// TIA Portal V16 export
// export: Created 2021-12-01T20:36:38.1325442Z, ExportSetting WithDefaults, DisplayName Totally Integrated Automation Portal, DisplayVersion V16 Update 4, DisplayName TIA Portal Version Control Interface, DisplayVersion V16 Update 2, DisplayName TIA Portal Openness, DisplayVersion V16 Update 4, DisplayName SINAMICS Startdrive Advanced, DisplayVersion V16 Update 5, DisplayName SINAMICS Startdrive G130, G150, S120, S150, SINAMICS MV, S210, DisplayVersion V16 Update 5, DisplayName SINAMICS Startdrive G110M, G120, G120C, G120D, G120P, G115D, DisplayVersion V16 Update 5, DisplayName STEP 7 Professional, DisplayVersion V16 Update 4, DisplayName STEP 7 Safety, DisplayVersion V16, DisplayName WinCC Advanced, DisplayVersion V16 Update 4
FUNCTION "ST00215_1_FC" : Void   // FC129, LAD
TITLE = ST00215_1
{ S7_Optimized_Access := 'TRUE' }
VERSION : 0.1
// stored: AutoNumber true, IsIECCheckEnabled false, SetENOAutomatically false, UDAEnableTagReadback false
   VAR_IN_OUT
      OPMODE : "OPMODE_OUT_UDT";
      HMI_EXTENSION : "HMI_EXTENSION_PANEL_UDT";
   END_VAR
   VAR_TEMP
      EmptyHS : "RT_HANDSHAKE_UDT";
   END_VAR
BEGIN

REGION Network 1: Alarm
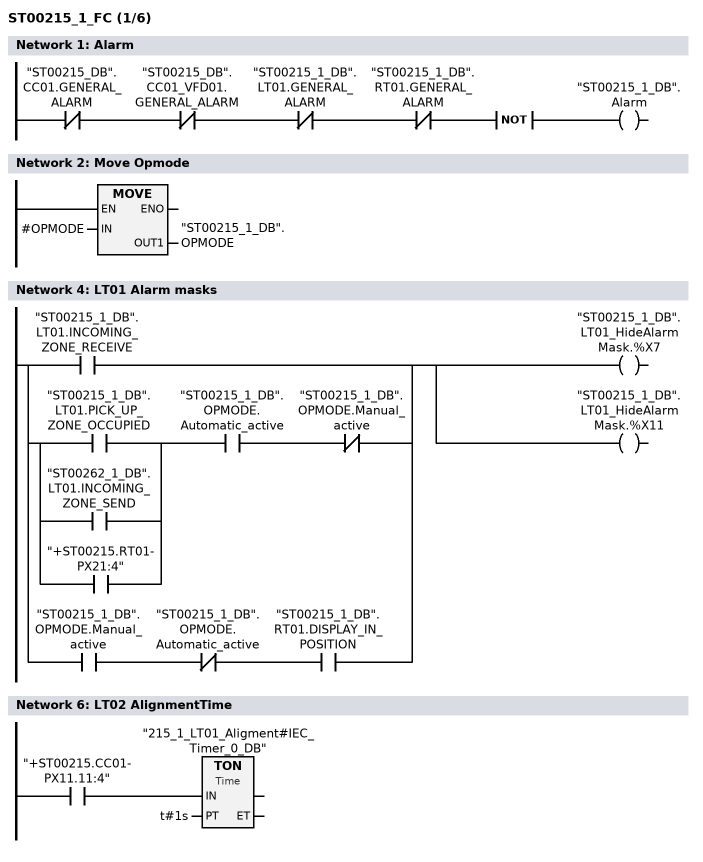
   RUNG wire#powerrail
      I_Contact( "ST00215_DB".CC01.GENERAL_ALARM )
      I_Contact( "ST00215_DB".CC01_VFD01.GENERAL_ALARM )
      I_Contact( "ST00215_1_DB".LT01.GENERAL_ALARM )
      I_Contact( "ST00215_1_DB".RT01.GENERAL_ALARM )
      Not()
      Coil( "ST00215_1_DB".Alarm )
   END_RUNG
   // the same network as SCL:
   "ST00215_1_DB".Alarm := NOT (NOT "ST00215_DB".CC01.GENERAL_ALARM AND NOT "ST00215_DB".CC01_VFD01.GENERAL_ALARM AND NOT "ST00215_1_DB".LT01.GENERAL_ALARM AND NOT "ST00215_1_DB".RT01.GENERAL_ALARM);
END_REGION

REGION Network 2: Move Opmode
   RUNG wire#powerrail
      Move(in := #OPMODE, out1 => "ST00215_1_DB".OPMODE)
   END_RUNG
   // the same network as SCL:
   "ST00215_1_DB".OPMODE := #OPMODE;
END_REGION

REGION Network 3: *******************LT01 Control*******************
END_REGION

REGION Network 4: LT01 Alarm masks
   RUNG wire#powerrail
      Contact( "ST00215_1_DB".LT01.INCOMING_ZONE_RECEIVE )
      wire#w1
      Coil( "ST00215_1_DB".LT01_HideAlarmMask.%X7 )
   END_RUNG
   RUNG wire#powerrail
      Contact( "ST00215_1_DB".LT01.PICK_UP_ZONE_OCCUPIED )
      wire#w2
      Contact( "ST00215_1_DB".OPMODE.Automatic_active )
      I_Contact( "ST00215_1_DB".OPMODE.Manual_active )
   END_RUNG wire#w1
   RUNG wire#powerrail
      Contact( "ST00262_1_DB".LT01.INCOMING_ZONE_SEND )
   END_RUNG wire#w2
   RUNG wire#powerrail
      Contact( "+ST00215.RT01-PX21:4" )
   END_RUNG wire#w2
   RUNG wire#powerrail
      Contact( "ST00215_1_DB".OPMODE.Manual_active )
      I_Contact( "ST00215_1_DB".OPMODE.Automatic_active )
      Contact( "ST00215_1_DB".RT01.DISPLAY_IN_POSITION )
   END_RUNG wire#w1
   RUNG wire#w1
      Coil( "ST00215_1_DB".LT01_HideAlarmMask.%X11 )
   END_RUNG
   // the same network as SCL:
   "ST00215_1_DB".LT01_HideAlarmMask.%X7 := "ST00215_1_DB".LT01.INCOMING_ZONE_RECEIVE OR (("ST00215_1_DB".LT01.PICK_UP_ZONE_OCCUPIED OR "ST00262_1_DB".LT01.INCOMING_ZONE_SEND OR "+ST00215.RT01-PX21:4") AND "ST00215_1_DB".OPMODE.Automatic_active AND NOT "ST00215_1_DB".OPMODE.Manual_active) OR ("ST00215_1_DB".OPMODE.Manual_active AND NOT "ST00215_1_DB".OPMODE.Automatic_active AND "ST00215_1_DB".RT01.DISPLAY_IN_POSITION);
   "ST00215_1_DB".LT01_HideAlarmMask.%X11 := "ST00215_1_DB".LT01_HideAlarmMask.%X7;
END_REGION

REGION Network 5 (SCL): LT01 Parameters
   "ST00215_1_DB".LT01.PARA_SET.Para.HasMidPosition := FALSE;
   "ST00215_1_DB".LT01.PARA_SET.Para.HasRT := true;
   "ST00215_1_DB".LT01.PARA_SET.Para.PosCCStopForward := true;
   "ST00215_1_DB".LT01.PARA_SET.Para.PosCCStopReverse := false;
   "ST00215_1_DB".LT01.PARA_SET.Para.PosRaiseForward_1 := true;
   "ST00215_1_DB".LT01.PARA_SET.Para.PosRaiseForward_2 := true;
   "ST00215_1_DB".LT01.PARA_SET.Para.PosRaiseReverse_1 := true;
   "ST00215_1_DB".LT01.PARA_SET.Para.PosRaiseReverse_2 := false;
   "ST00215_1_DB".LT01.PARA_SET.Para.PosSlowForward := true;
   "ST00215_1_DB".LT01.PARA_SET.Para.PosSlowReverse := false;
   "ST00215_1_DB".LT01.PARA_SET.Set.RuntimeLower := t#10s;
   "ST00215_1_DB".LT01.PARA_SET.Set.RuntimeLift := t#11s;
   "ST00215_1_DB".LT01.PARA_SET.Set.AlignmentTime := t#0ms;
END_REGION

REGION Network 6: LT02 AlignmentTime
   RUNG wire#powerrail
      Contact( "+ST00215.CC01-PX11.11:4" )
      { S7_Templates := "time_type := Time" } "215_1_LT01_Aligment#IEC_Timer_0_DB".TON(pt := t#1s, et =>)
   END_RUNG
   // the same network as SCL:
   "215_1_LT01_Aligment#IEC_Timer_0_DB".TON(IN := "+ST00215.CC01-PX11.11:4", PT := t#1s);
END_REGION

REGION Network 7: LT01 CC Place FB
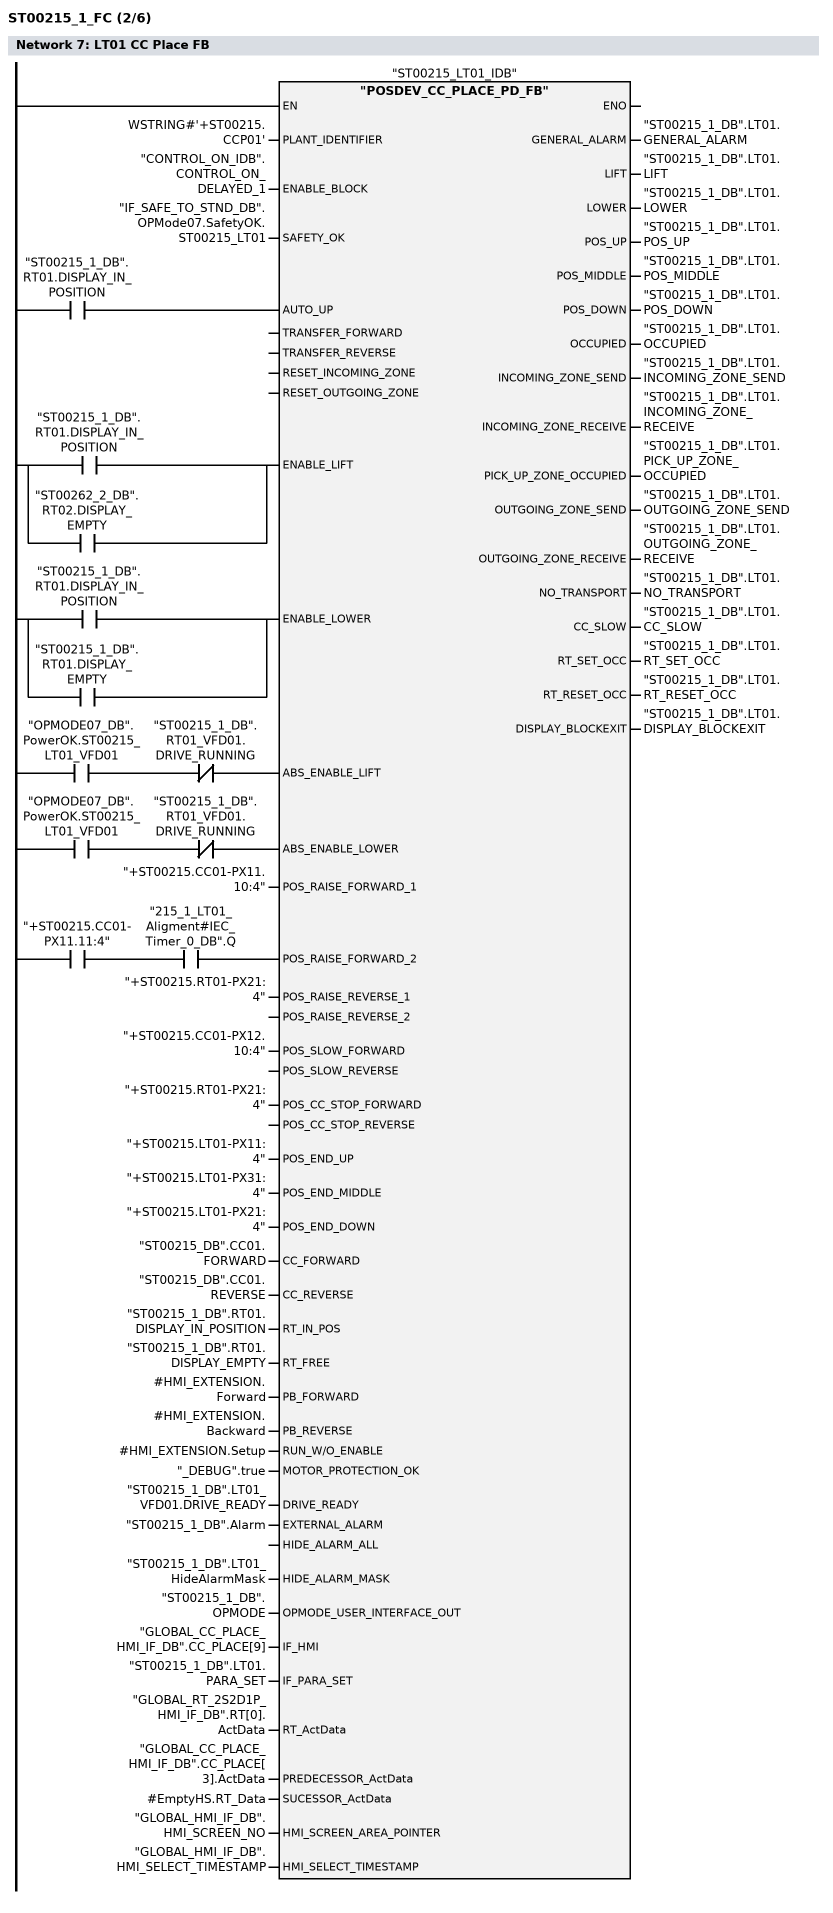
   RUNG wire#powerrail
      "ST00215_LT01_IDB"(AUTO_UP := wire#w1, ENABLE_LIFT := wire#w2, ENABLE_LOWER := wire#w3, ABS_ENABLE_LIFT := wire#w4, ABS_ENABLE_LOWER := wire#w5, POS_RAISE_FORWARD_2 := wire#w6, PLANT_IDENTIFIER := WSTRING#'+ST00215.CCP01', ENABLE_BLOCK := "CONTROL_ON_IDB".CONTROL_ON_DELAYED_1, SAFETY_OK := "IF_SAFE_TO_STND_DB".OPMode07.SafetyOK.ST00215_LT01, TRANSFER_FORWARD :=, TRANSFER_REVERSE :=, RESET_INCOMING_ZONE :=, RESET_OUTGOING_ZONE :=, POS_RAISE_FORWARD_1 := "+ST00215.CC01-PX11.10:4", POS_RAISE_REVERSE_1 := "+ST00215.RT01-PX21:4", POS_RAISE_REVERSE_2 :=, POS_SLOW_FORWARD := "+ST00215.CC01-PX12.10:4", POS_SLOW_REVERSE :=, POS_CC_STOP_FORWARD := "+ST00215.RT01-PX21:4", POS_CC_STOP_REVERSE :=, POS_END_UP := "+ST00215.LT01-PX11:4", POS_END_MIDDLE := "+ST00215.LT01-PX31:4", POS_END_DOWN := "+ST00215.LT01-PX21:4", CC_FORWARD := "ST00215_DB".CC01.FORWARD, CC_REVERSE := "ST00215_DB".CC01.REVERSE, RT_IN_POS := "ST00215_1_DB".RT01.DISPLAY_IN_POSITION, RT_FREE := "ST00215_1_DB".RT01.DISPLAY_EMPTY, PB_FORWARD := #HMI_EXTENSION.Forward, PB_REVERSE := #HMI_EXTENSION.Backward, "RUN_W/O_ENABLE" := #HMI_EXTENSION.Setup, MOTOR_PROTECTION_OK := "_DEBUG".true, DRIVE_READY := "ST00215_1_DB".LT01_VFD01.DRIVE_READY, EXTERNAL_ALARM := "ST00215_1_DB".Alarm, HIDE_ALARM_ALL :=, HIDE_ALARM_MASK := "ST00215_1_DB".LT01_HideAlarmMask, OPMODE_USER_INTERFACE_OUT := "ST00215_1_DB".OPMODE, IF_HMI := "GLOBAL_CC_PLACE_HMI_IF_DB".CC_PLACE[9], IF_PARA_SET := "ST00215_1_DB".LT01.PARA_SET, RT_ActData := "GLOBAL_RT_2S2D1P_HMI_IF_DB".RT[0].ActData, PREDECESSOR_ActData := "GLOBAL_CC_PLACE_HMI_IF_DB".CC_PLACE[3].ActData, SUCESSOR_ActData := #EmptyHS.RT_Data, HMI_SCREEN_AREA_POINTER := "GLOBAL_HMI_IF_DB".HMI_SCREEN_NO, HMI_SELECT_TIMESTAMP := "GLOBAL_HMI_IF_DB".HMI_SELECT_TIMESTAMP, GENERAL_ALARM => "ST00215_1_DB".LT01.GENERAL_ALARM, LIFT => "ST00215_1_DB".LT01.LIFT, LOWER => "ST00215_1_DB".LT01.LOWER, POS_UP => "ST00215_1_DB".LT01.POS_UP, POS_MIDDLE => "ST00215_1_DB".LT01.POS_MIDDLE, POS_DOWN => "ST00215_1_DB".LT01.POS_DOWN, OCCUPIED => "ST00215_1_DB".LT01.OCCUPIED, INCOMING_ZONE_SEND => "ST00215_1_DB".LT01.INCOMING_ZONE_SEND, INCOMING_ZONE_RECEIVE => "ST00215_1_DB".LT01.INCOMING_ZONE_RECEIVE, PICK_UP_ZONE_OCCUPIED => "ST00215_1_DB".LT01.PICK_UP_ZONE_OCCUPIED, OUTGOING_ZONE_SEND => "ST00215_1_DB".LT01.OUTGOING_ZONE_SEND, OUTGOING_ZONE_RECEIVE => "ST00215_1_DB".LT01.OUTGOING_ZONE_RECEIVE, NO_TRANSPORT => "ST00215_1_DB".LT01.NO_TRANSPORT, CC_SLOW => "ST00215_1_DB".LT01.CC_SLOW, RT_SET_OCC => "ST00215_1_DB".LT01.RT_SET_OCC, RT_RESET_OCC => "ST00215_1_DB".LT01.RT_RESET_OCC, DISPLAY_BLOCKEXIT => "ST00215_1_DB".LT01.DISPLAY_BLOCKEXIT)
   END_RUNG
   RUNG wire#powerrail
      Contact( "ST00215_1_DB".RT01.DISPLAY_IN_POSITION )
   END_RUNG wire#w1
   RUNG wire#powerrail
      Contact( "ST00215_1_DB".RT01.DISPLAY_IN_POSITION )
   END_RUNG wire#w2
   RUNG wire#powerrail
      Contact( "ST00262_2_DB".RT02.DISPLAY_EMPTY )
   END_RUNG wire#w2
   RUNG wire#powerrail
      Contact( "ST00215_1_DB".RT01.DISPLAY_IN_POSITION )
   END_RUNG wire#w3
   RUNG wire#powerrail
      Contact( "ST00215_1_DB".RT01.DISPLAY_EMPTY )
   END_RUNG wire#w3
   RUNG wire#powerrail
      Contact( "OPMODE07_DB".PowerOK.ST00215_LT01_VFD01 )
      I_Contact( "ST00215_1_DB".RT01_VFD01.DRIVE_RUNNING )
   END_RUNG wire#w4
   RUNG wire#powerrail
      Contact( "OPMODE07_DB".PowerOK.ST00215_LT01_VFD01 )
      I_Contact( "ST00215_1_DB".RT01_VFD01.DRIVE_RUNNING )
   END_RUNG wire#w5
   RUNG wire#powerrail
      Contact( "+ST00215.CC01-PX11.11:4" )
      Contact( "215_1_LT01_Aligment#IEC_Timer_0_DB".Q )
   END_RUNG wire#w6
   // the same network as SCL:
   "ST00215_LT01_IDB"(PLANT_IDENTIFIER := WSTRING#'+ST00215.CCP01',   // "POSDEV_CC_PLACE_PD_FB"
                      ENABLE_BLOCK := "CONTROL_ON_IDB".CONTROL_ON_DELAYED_1,
                      SAFETY_OK := "IF_SAFE_TO_STND_DB".OPMode07.SafetyOK.ST00215_LT01,
                      AUTO_UP := "ST00215_1_DB".RT01.DISPLAY_IN_POSITION,
                      ENABLE_LIFT := "ST00215_1_DB".RT01.DISPLAY_IN_POSITION OR "ST00262_2_DB".RT02.DISPLAY_EMPTY,
                      ENABLE_LOWER := "ST00215_1_DB".RT01.DISPLAY_IN_POSITION OR "ST00215_1_DB".RT01.DISPLAY_EMPTY,
                      ABS_ENABLE_LIFT := "OPMODE07_DB".PowerOK.ST00215_LT01_VFD01 AND NOT "ST00215_1_DB".RT01_VFD01.DRIVE_RUNNING,
                      ABS_ENABLE_LOWER := "OPMODE07_DB".PowerOK.ST00215_LT01_VFD01 AND NOT "ST00215_1_DB".RT01_VFD01.DRIVE_RUNNING,
                      POS_RAISE_FORWARD_1 := "+ST00215.CC01-PX11.10:4",
                      POS_RAISE_FORWARD_2 := "+ST00215.CC01-PX11.11:4" AND "215_1_LT01_Aligment#IEC_Timer_0_DB".Q,
                      POS_RAISE_REVERSE_1 := "+ST00215.RT01-PX21:4",
                      POS_SLOW_FORWARD := "+ST00215.CC01-PX12.10:4",
                      POS_CC_STOP_FORWARD := "+ST00215.RT01-PX21:4",
                      POS_END_UP := "+ST00215.LT01-PX11:4",
                      POS_END_MIDDLE := "+ST00215.LT01-PX31:4",
                      POS_END_DOWN := "+ST00215.LT01-PX21:4",
                      CC_FORWARD := "ST00215_DB".CC01.FORWARD,
                      CC_REVERSE := "ST00215_DB".CC01.REVERSE,
                      RT_IN_POS := "ST00215_1_DB".RT01.DISPLAY_IN_POSITION,
                      RT_FREE := "ST00215_1_DB".RT01.DISPLAY_EMPTY,
                      PB_FORWARD := #HMI_EXTENSION.Forward,
                      PB_REVERSE := #HMI_EXTENSION.Backward,
                      "RUN_W/O_ENABLE" := #HMI_EXTENSION.Setup,
                      MOTOR_PROTECTION_OK := "_DEBUG".true,
                      DRIVE_READY := "ST00215_1_DB".LT01_VFD01.DRIVE_READY,
                      EXTERNAL_ALARM := "ST00215_1_DB".Alarm,
                      HIDE_ALARM_MASK := "ST00215_1_DB".LT01_HideAlarmMask,
                      OPMODE_USER_INTERFACE_OUT := "ST00215_1_DB".OPMODE,
                      IF_HMI := "GLOBAL_CC_PLACE_HMI_IF_DB".CC_PLACE[9],
                      IF_PARA_SET := "ST00215_1_DB".LT01.PARA_SET,
                      RT_ActData := "GLOBAL_RT_2S2D1P_HMI_IF_DB".RT[0].ActData,
                      PREDECESSOR_ActData := "GLOBAL_CC_PLACE_HMI_IF_DB".CC_PLACE[3].ActData,
                      SUCESSOR_ActData := #EmptyHS.RT_Data,
                      HMI_SCREEN_AREA_POINTER := "GLOBAL_HMI_IF_DB".HMI_SCREEN_NO,
                      HMI_SELECT_TIMESTAMP := "GLOBAL_HMI_IF_DB".HMI_SELECT_TIMESTAMP,
                      GENERAL_ALARM => "ST00215_1_DB".LT01.GENERAL_ALARM,
                      LIFT => "ST00215_1_DB".LT01.LIFT,
                      LOWER => "ST00215_1_DB".LT01.LOWER,
                      POS_UP => "ST00215_1_DB".LT01.POS_UP,
                      POS_MIDDLE => "ST00215_1_DB".LT01.POS_MIDDLE,
                      POS_DOWN => "ST00215_1_DB".LT01.POS_DOWN,
                      OCCUPIED => "ST00215_1_DB".LT01.OCCUPIED,
                      INCOMING_ZONE_SEND => "ST00215_1_DB".LT01.INCOMING_ZONE_SEND,
                      INCOMING_ZONE_RECEIVE => "ST00215_1_DB".LT01.INCOMING_ZONE_RECEIVE,
                      PICK_UP_ZONE_OCCUPIED => "ST00215_1_DB".LT01.PICK_UP_ZONE_OCCUPIED,
                      OUTGOING_ZONE_SEND => "ST00215_1_DB".LT01.OUTGOING_ZONE_SEND,
                      OUTGOING_ZONE_RECEIVE => "ST00215_1_DB".LT01.OUTGOING_ZONE_RECEIVE,
                      NO_TRANSPORT => "ST00215_1_DB".LT01.NO_TRANSPORT,
                      CC_SLOW => "ST00215_1_DB".LT01.CC_SLOW,
                      RT_SET_OCC => "ST00215_1_DB".LT01.RT_SET_OCC,
                      RT_RESET_OCC => "ST00215_1_DB".LT01.RT_RESET_OCC,
                      DISPLAY_BLOCKEXIT => "ST00215_1_DB".LT01.DISPLAY_BLOCKEXIT);
END_REGION

REGION Network 8: LT01 Speed
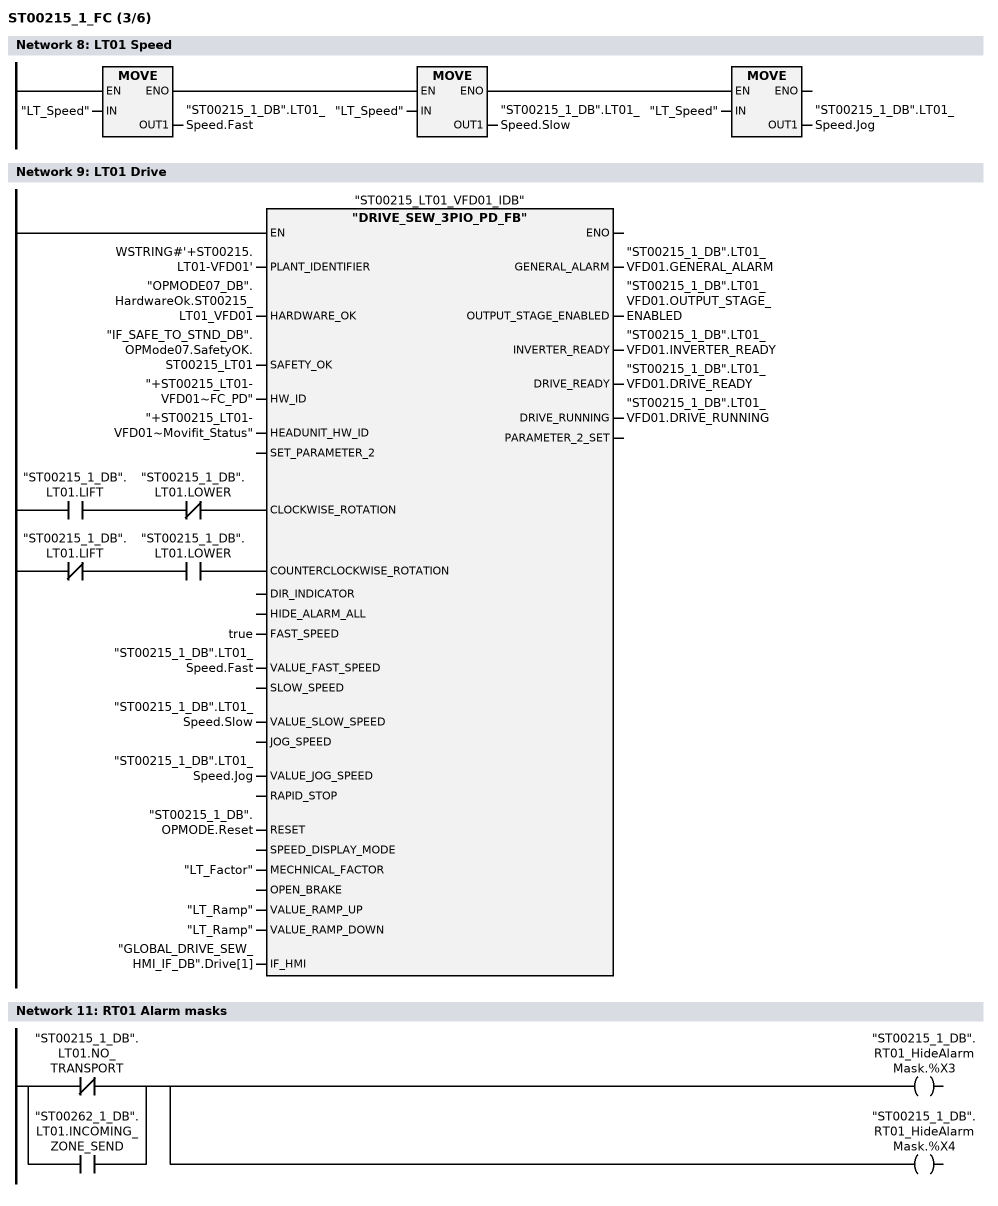
   RUNG wire#powerrail
      Move(in := "LT_Speed", out1 => "ST00215_1_DB".LT01_Speed.Fast)
      Move(in := "LT_Speed", out1 => "ST00215_1_DB".LT01_Speed.Slow)
      Move(in := "LT_Speed", out1 => "ST00215_1_DB".LT01_Speed.Jog)
   END_RUNG
   // the same network as SCL:
   "ST00215_1_DB".LT01_Speed.Fast := "LT_Speed";
   "ST00215_1_DB".LT01_Speed.Slow := "LT_Speed";
   "ST00215_1_DB".LT01_Speed.Jog := "LT_Speed";
END_REGION

REGION Network 9: LT01 Drive
   RUNG wire#powerrail
      "ST00215_LT01_VFD01_IDB"(CLOCKWISE_ROTATION := wire#w1, COUNTERCLOCKWISE_ROTATION := wire#w2, PLANT_IDENTIFIER := WSTRING#'+ST00215.LT01-VFD01', HARDWARE_OK := "OPMODE07_DB".HardwareOk.ST00215_LT01_VFD01, SAFETY_OK := "IF_SAFE_TO_STND_DB".OPMode07.SafetyOK.ST00215_LT01, HW_ID := "+ST00215_LT01-VFD01~FC_PD", HEADUNIT_HW_ID := "+ST00215_LT01-VFD01~Movifit_Status", SET_PARAMETER_2 :=, DIR_INDICATOR :=, HIDE_ALARM_ALL :=, FAST_SPEED := true, VALUE_FAST_SPEED := "ST00215_1_DB".LT01_Speed.Fast, SLOW_SPEED :=, VALUE_SLOW_SPEED := "ST00215_1_DB".LT01_Speed.Slow, JOG_SPEED :=, VALUE_JOG_SPEED := "ST00215_1_DB".LT01_Speed.Jog, RAPID_STOP :=, RESET := "ST00215_1_DB".OPMODE.Reset, SPEED_DISPLAY_MODE :=, MECHNICAL_FACTOR := "LT_Factor", OPEN_BRAKE :=, VALUE_RAMP_UP := "LT_Ramp", VALUE_RAMP_DOWN := "LT_Ramp", IF_HMI := "GLOBAL_DRIVE_SEW_HMI_IF_DB".Drive[1], GENERAL_ALARM => "ST00215_1_DB".LT01_VFD01.GENERAL_ALARM, OUTPUT_STAGE_ENABLED => "ST00215_1_DB".LT01_VFD01.OUTPUT_STAGE_ENABLED, INVERTER_READY => "ST00215_1_DB".LT01_VFD01.INVERTER_READY, DRIVE_READY => "ST00215_1_DB".LT01_VFD01.DRIVE_READY, DRIVE_RUNNING => "ST00215_1_DB".LT01_VFD01.DRIVE_RUNNING, PARAMETER_2_SET =>)
   END_RUNG
   RUNG wire#powerrail
      Contact( "ST00215_1_DB".LT01.LIFT )
      I_Contact( "ST00215_1_DB".LT01.LOWER )
   END_RUNG wire#w1
   RUNG wire#powerrail
      I_Contact( "ST00215_1_DB".LT01.LIFT )
      Contact( "ST00215_1_DB".LT01.LOWER )
   END_RUNG wire#w2
   // the same network as SCL:
   "ST00215_LT01_VFD01_IDB"(PLANT_IDENTIFIER := WSTRING#'+ST00215.LT01-VFD01',   // "DRIVE_SEW_3PIO_PD_FB"
                           HARDWARE_OK := "OPMODE07_DB".HardwareOk.ST00215_LT01_VFD01,
                           SAFETY_OK := "IF_SAFE_TO_STND_DB".OPMode07.SafetyOK.ST00215_LT01,
                           HW_ID := "+ST00215_LT01-VFD01~FC_PD",
                           HEADUNIT_HW_ID := "+ST00215_LT01-VFD01~Movifit_Status",
                           CLOCKWISE_ROTATION := "ST00215_1_DB".LT01.LIFT AND NOT "ST00215_1_DB".LT01.LOWER,
                           COUNTERCLOCKWISE_ROTATION := NOT "ST00215_1_DB".LT01.LIFT AND "ST00215_1_DB".LT01.LOWER,
                           FAST_SPEED := true,
                           VALUE_FAST_SPEED := "ST00215_1_DB".LT01_Speed.Fast,
                           VALUE_SLOW_SPEED := "ST00215_1_DB".LT01_Speed.Slow,
                           VALUE_JOG_SPEED := "ST00215_1_DB".LT01_Speed.Jog,
                           RESET := "ST00215_1_DB".OPMODE.Reset,
                           MECHNICAL_FACTOR := "LT_Factor",
                           VALUE_RAMP_UP := "LT_Ramp",
                           VALUE_RAMP_DOWN := "LT_Ramp",
                           IF_HMI := "GLOBAL_DRIVE_SEW_HMI_IF_DB".Drive[1],
                           GENERAL_ALARM => "ST00215_1_DB".LT01_VFD01.GENERAL_ALARM,
                           OUTPUT_STAGE_ENABLED => "ST00215_1_DB".LT01_VFD01.OUTPUT_STAGE_ENABLED,
                           INVERTER_READY => "ST00215_1_DB".LT01_VFD01.INVERTER_READY,
                           DRIVE_READY => "ST00215_1_DB".LT01_VFD01.DRIVE_READY,
                           DRIVE_RUNNING => "ST00215_1_DB".LT01_VFD01.DRIVE_RUNNING);
END_REGION

REGION Network 10: *******************RT01 Control*******************
END_REGION

REGION Network 11: RT01 Alarm masks
   RUNG wire#powerrail
      I_Contact( "ST00215_1_DB".LT01.NO_TRANSPORT )
      wire#w1
      Coil( "ST00215_1_DB".RT01_HideAlarmMask.%X3 )
   END_RUNG
   RUNG wire#powerrail
      Contact( "ST00262_1_DB".LT01.INCOMING_ZONE_SEND )
   END_RUNG wire#w1
   RUNG wire#w1
      Coil( "ST00215_1_DB".RT01_HideAlarmMask.%X4 )
   END_RUNG
   // the same network as SCL:
   "ST00215_1_DB".RT01_HideAlarmMask.%X3 := NOT "ST00215_1_DB".LT01.NO_TRANSPORT OR "ST00262_1_DB".LT01.INCOMING_ZONE_SEND;
   "ST00215_1_DB".RT01_HideAlarmMask.%X4 := "ST00215_1_DB".RT01_HideAlarmMask.%X3;
END_REGION

REGION Network 12 (SCL): RT01 Parameters
   "ST00215_1_DB".RT01.PARA_SET.Para.PosEndForward1 := true;
   "ST00215_1_DB".RT01.PARA_SET.Para.PosEndReverse := true;
   "ST00215_1_DB".RT01.PARA_SET.Para.PosSlowForward := true;

   "ST00215_1_DB".RT01.PARA_SET.Set.RunTimeForward := 450;
   "ST00215_1_DB".RT01.PARA_SET.Set.RunTimeReverse := 450;
END_REGION

REGION Network 13: RT01 HandShake
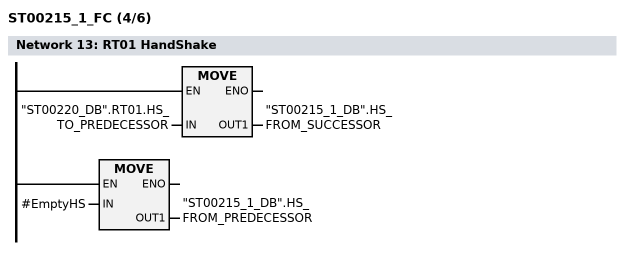
   RUNG wire#powerrail
      Move(in := "ST00220_DB".RT01.HS_TO_PREDECESSOR, out1 => "ST00215_1_DB".HS_FROM_SUCCESSOR)
   END_RUNG
   RUNG wire#powerrail
      Move(in := #EmptyHS, out1 => "ST00215_1_DB".HS_FROM_PREDECESSOR)
   END_RUNG
   // the same network as SCL:
   "ST00215_1_DB".HS_FROM_SUCCESSOR := "ST00220_DB".RT01.HS_TO_PREDECESSOR;
   "ST00215_1_DB".HS_FROM_PREDECESSOR := #EmptyHS;
END_REGION

REGION Network 14: RT01 FB Control
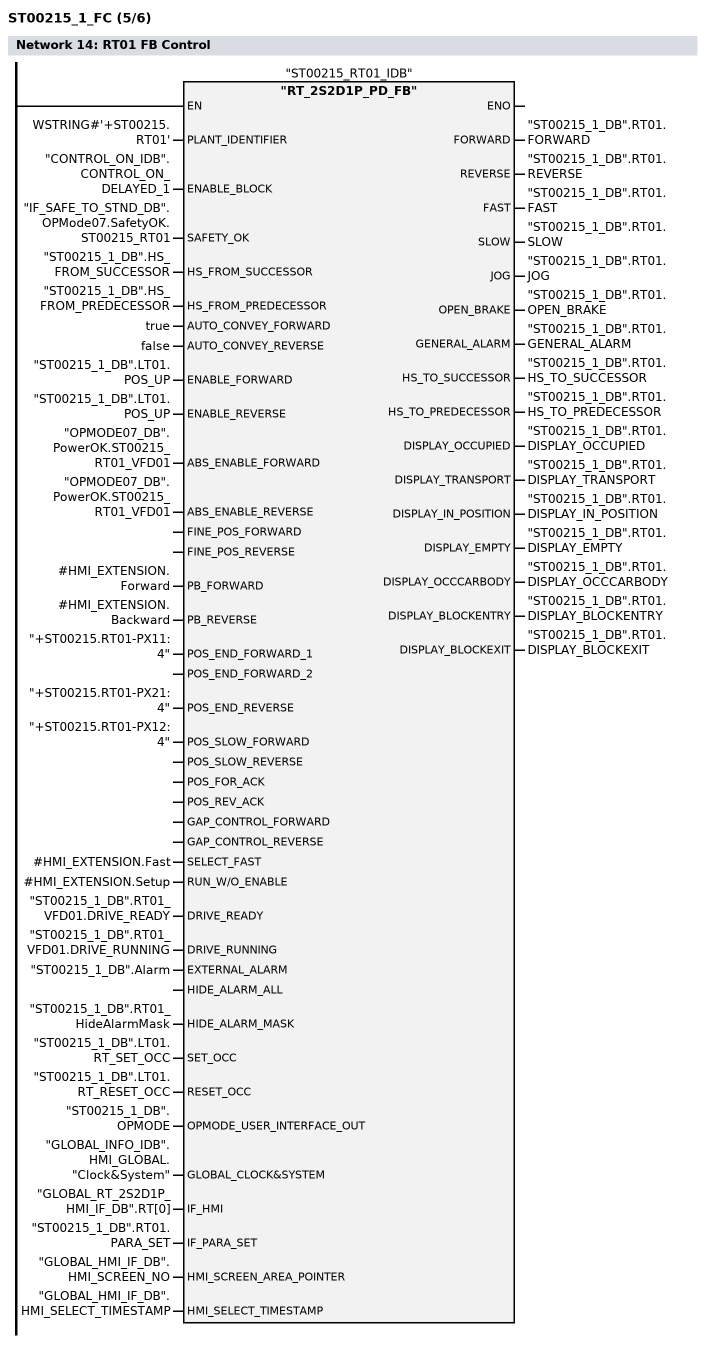
   RUNG wire#powerrail
      "ST00215_RT01_IDB"(PLANT_IDENTIFIER := WSTRING#'+ST00215.RT01', ENABLE_BLOCK := "CONTROL_ON_IDB".CONTROL_ON_DELAYED_1, SAFETY_OK := "IF_SAFE_TO_STND_DB".OPMode07.SafetyOK.ST00215_RT01, HS_FROM_SUCCESSOR := "ST00215_1_DB".HS_FROM_SUCCESSOR, HS_FROM_PREDECESSOR := "ST00215_1_DB".HS_FROM_PREDECESSOR, AUTO_CONVEY_FORWARD := true, AUTO_CONVEY_REVERSE := false, ENABLE_FORWARD := "ST00215_1_DB".LT01.POS_UP, ENABLE_REVERSE := "ST00215_1_DB".LT01.POS_UP, ABS_ENABLE_FORWARD := "OPMODE07_DB".PowerOK.ST00215_RT01_VFD01, ABS_ENABLE_REVERSE := "OPMODE07_DB".PowerOK.ST00215_RT01_VFD01, FINE_POS_FORWARD :=, FINE_POS_REVERSE :=, PB_FORWARD := #HMI_EXTENSION.Forward, PB_REVERSE := #HMI_EXTENSION.Backward, POS_END_FORWARD_1 := "+ST00215.RT01-PX11:4", POS_END_FORWARD_2 :=, POS_END_REVERSE := "+ST00215.RT01-PX21:4", POS_SLOW_FORWARD := "+ST00215.RT01-PX12:4", POS_SLOW_REVERSE :=, POS_FOR_ACK :=, POS_REV_ACK :=, GAP_CONTROL_FORWARD :=, GAP_CONTROL_REVERSE :=, SELECT_FAST := #HMI_EXTENSION.Fast, "RUN_W/O_ENABLE" := #HMI_EXTENSION.Setup, DRIVE_READY := "ST00215_1_DB".RT01_VFD01.DRIVE_READY, DRIVE_RUNNING := "ST00215_1_DB".RT01_VFD01.DRIVE_RUNNING, EXTERNAL_ALARM := "ST00215_1_DB".Alarm, HIDE_ALARM_ALL :=, HIDE_ALARM_MASK := "ST00215_1_DB".RT01_HideAlarmMask, SET_OCC := "ST00215_1_DB".LT01.RT_SET_OCC, RESET_OCC := "ST00215_1_DB".LT01.RT_RESET_OCC, OPMODE_USER_INTERFACE_OUT := "ST00215_1_DB".OPMODE, "GLOBAL_CLOCK&SYSTEM" := "GLOBAL_INFO_IDB".HMI_GLOBAL."Clock&System", IF_HMI := "GLOBAL_RT_2S2D1P_HMI_IF_DB".RT[0], IF_PARA_SET := "ST00215_1_DB".RT01.PARA_SET, HMI_SCREEN_AREA_POINTER := "GLOBAL_HMI_IF_DB".HMI_SCREEN_NO, HMI_SELECT_TIMESTAMP := "GLOBAL_HMI_IF_DB".HMI_SELECT_TIMESTAMP, FORWARD => "ST00215_1_DB".RT01.FORWARD, REVERSE => "ST00215_1_DB".RT01.REVERSE, FAST => "ST00215_1_DB".RT01.FAST, SLOW => "ST00215_1_DB".RT01.SLOW, JOG => "ST00215_1_DB".RT01.JOG, OPEN_BRAKE => "ST00215_1_DB".RT01.OPEN_BRAKE, GENERAL_ALARM => "ST00215_1_DB".RT01.GENERAL_ALARM, HS_TO_SUCCESSOR => "ST00215_1_DB".RT01.HS_TO_SUCCESSOR, HS_TO_PREDECESSOR => "ST00215_1_DB".RT01.HS_TO_PREDECESSOR, DISPLAY_OCCUPIED => "ST00215_1_DB".RT01.DISPLAY_OCCUPIED, DISPLAY_TRANSPORT => "ST00215_1_DB".RT01.DISPLAY_TRANSPORT, DISPLAY_IN_POSITION => "ST00215_1_DB".RT01.DISPLAY_IN_POSITION, DISPLAY_EMPTY => "ST00215_1_DB".RT01.DISPLAY_EMPTY, DISPLAY_OCCCARBODY => "ST00215_1_DB".RT01.DISPLAY_OCCCARBODY, DISPLAY_BLOCKENTRY => "ST00215_1_DB".RT01.DISPLAY_BLOCKENTRY, DISPLAY_BLOCKEXIT => "ST00215_1_DB".RT01.DISPLAY_BLOCKEXIT)
   END_RUNG
   // the same network as SCL:
   "ST00215_RT01_IDB"(PLANT_IDENTIFIER := WSTRING#'+ST00215.RT01',   // "RT_2S2D1P_PD_FB"
                      ENABLE_BLOCK := "CONTROL_ON_IDB".CONTROL_ON_DELAYED_1,
                      SAFETY_OK := "IF_SAFE_TO_STND_DB".OPMode07.SafetyOK.ST00215_RT01,
                      HS_FROM_SUCCESSOR := "ST00215_1_DB".HS_FROM_SUCCESSOR,
                      HS_FROM_PREDECESSOR := "ST00215_1_DB".HS_FROM_PREDECESSOR,
                      AUTO_CONVEY_FORWARD := true,
                      AUTO_CONVEY_REVERSE := false,
                      ENABLE_FORWARD := "ST00215_1_DB".LT01.POS_UP,
                      ENABLE_REVERSE := "ST00215_1_DB".LT01.POS_UP,
                      ABS_ENABLE_FORWARD := "OPMODE07_DB".PowerOK.ST00215_RT01_VFD01,
                      ABS_ENABLE_REVERSE := "OPMODE07_DB".PowerOK.ST00215_RT01_VFD01,
                      PB_FORWARD := #HMI_EXTENSION.Forward,
                      PB_REVERSE := #HMI_EXTENSION.Backward,
                      POS_END_FORWARD_1 := "+ST00215.RT01-PX11:4",
                      POS_END_REVERSE := "+ST00215.RT01-PX21:4",
                      POS_SLOW_FORWARD := "+ST00215.RT01-PX12:4",
                      SELECT_FAST := #HMI_EXTENSION.Fast,
                      "RUN_W/O_ENABLE" := #HMI_EXTENSION.Setup,
                      DRIVE_READY := "ST00215_1_DB".RT01_VFD01.DRIVE_READY,
                      DRIVE_RUNNING := "ST00215_1_DB".RT01_VFD01.DRIVE_RUNNING,
                      EXTERNAL_ALARM := "ST00215_1_DB".Alarm,
                      HIDE_ALARM_MASK := "ST00215_1_DB".RT01_HideAlarmMask,
                      SET_OCC := "ST00215_1_DB".LT01.RT_SET_OCC,
                      RESET_OCC := "ST00215_1_DB".LT01.RT_RESET_OCC,
                      OPMODE_USER_INTERFACE_OUT := "ST00215_1_DB".OPMODE,
                      "GLOBAL_CLOCK&SYSTEM" := "GLOBAL_INFO_IDB".HMI_GLOBAL."Clock&System",
                      IF_HMI := "GLOBAL_RT_2S2D1P_HMI_IF_DB".RT[0],
                      IF_PARA_SET := "ST00215_1_DB".RT01.PARA_SET,
                      HMI_SCREEN_AREA_POINTER := "GLOBAL_HMI_IF_DB".HMI_SCREEN_NO,
                      HMI_SELECT_TIMESTAMP := "GLOBAL_HMI_IF_DB".HMI_SELECT_TIMESTAMP,
                      FORWARD => "ST00215_1_DB".RT01.FORWARD,
                      REVERSE => "ST00215_1_DB".RT01.REVERSE,
                      FAST => "ST00215_1_DB".RT01.FAST,
                      SLOW => "ST00215_1_DB".RT01.SLOW,
                      JOG => "ST00215_1_DB".RT01.JOG,
                      OPEN_BRAKE => "ST00215_1_DB".RT01.OPEN_BRAKE,
                      GENERAL_ALARM => "ST00215_1_DB".RT01.GENERAL_ALARM,
                      HS_TO_SUCCESSOR => "ST00215_1_DB".RT01.HS_TO_SUCCESSOR,
                      HS_TO_PREDECESSOR => "ST00215_1_DB".RT01.HS_TO_PREDECESSOR,
                      DISPLAY_OCCUPIED => "ST00215_1_DB".RT01.DISPLAY_OCCUPIED,
                      DISPLAY_TRANSPORT => "ST00215_1_DB".RT01.DISPLAY_TRANSPORT,
                      DISPLAY_IN_POSITION => "ST00215_1_DB".RT01.DISPLAY_IN_POSITION,
                      DISPLAY_EMPTY => "ST00215_1_DB".RT01.DISPLAY_EMPTY,
                      DISPLAY_OCCCARBODY => "ST00215_1_DB".RT01.DISPLAY_OCCCARBODY,
                      DISPLAY_BLOCKENTRY => "ST00215_1_DB".RT01.DISPLAY_BLOCKENTRY,
                      DISPLAY_BLOCKEXIT => "ST00215_1_DB".RT01.DISPLAY_BLOCKEXIT);
END_REGION

REGION Network 15: RT01 Speed
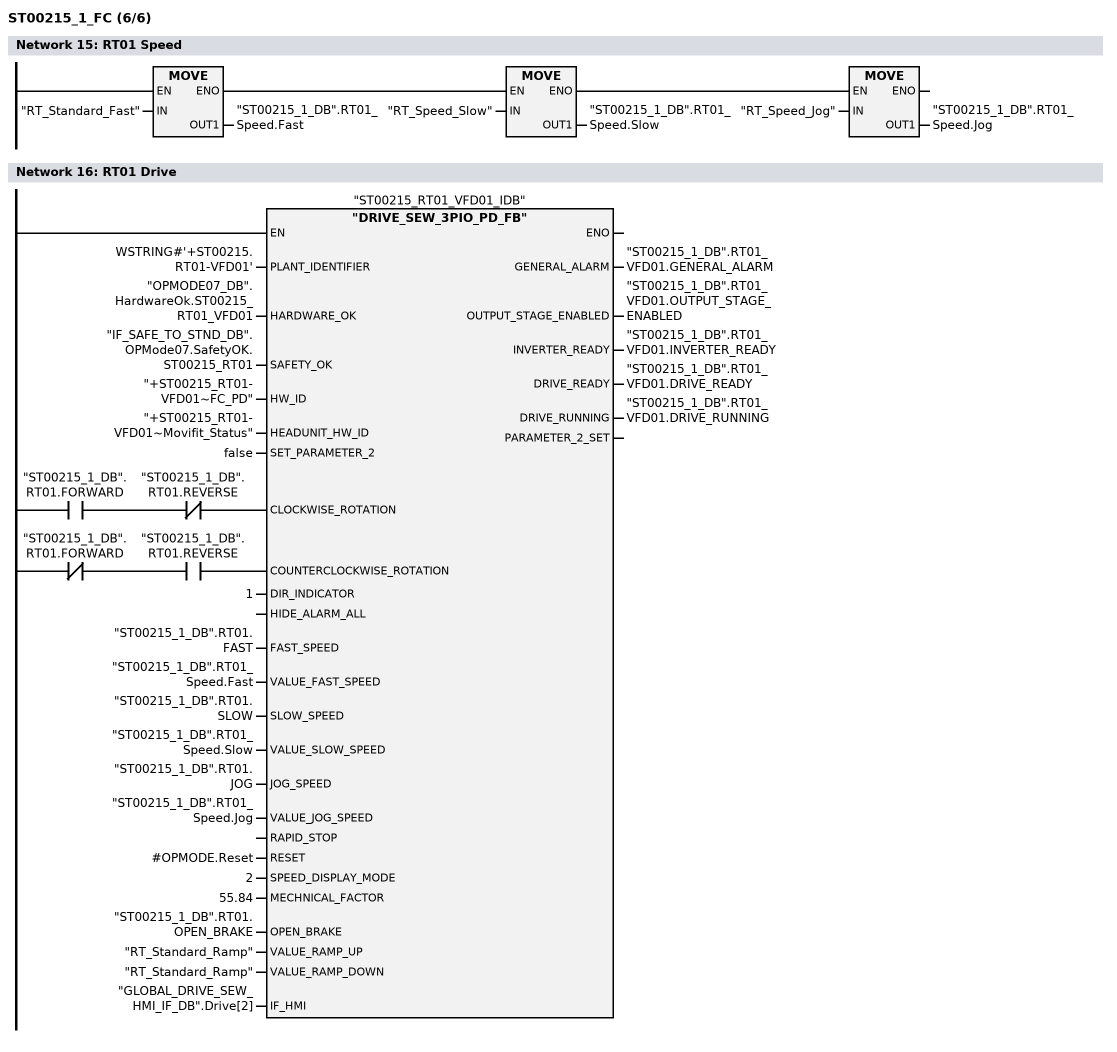
   RUNG wire#powerrail
      Move(in := "RT_Standard_Fast", out1 => "ST00215_1_DB".RT01_Speed.Fast)
      Move(in := "RT_Speed_Slow", out1 => "ST00215_1_DB".RT01_Speed.Slow)
      Move(in := "RT_Speed_Jog", out1 => "ST00215_1_DB".RT01_Speed.Jog)
   END_RUNG
   // the same network as SCL:
   "ST00215_1_DB".RT01_Speed.Fast := "RT_Standard_Fast";
   "ST00215_1_DB".RT01_Speed.Slow := "RT_Speed_Slow";
   "ST00215_1_DB".RT01_Speed.Jog := "RT_Speed_Jog";
END_REGION

REGION Network 16: RT01 Drive
   RUNG wire#powerrail
      "ST00215_RT01_VFD01_IDB"(CLOCKWISE_ROTATION := wire#w1, COUNTERCLOCKWISE_ROTATION := wire#w2, PLANT_IDENTIFIER := WSTRING#'+ST00215.RT01-VFD01', HARDWARE_OK := "OPMODE07_DB".HardwareOk.ST00215_RT01_VFD01, SAFETY_OK := "IF_SAFE_TO_STND_DB".OPMode07.SafetyOK.ST00215_RT01, HW_ID := "+ST00215_RT01-VFD01~FC_PD", HEADUNIT_HW_ID := "+ST00215_RT01-VFD01~Movifit_Status", SET_PARAMETER_2 := false, DIR_INDICATOR := 1, HIDE_ALARM_ALL :=, FAST_SPEED := "ST00215_1_DB".RT01.FAST, VALUE_FAST_SPEED := "ST00215_1_DB".RT01_Speed.Fast, SLOW_SPEED := "ST00215_1_DB".RT01.SLOW, VALUE_SLOW_SPEED := "ST00215_1_DB".RT01_Speed.Slow, JOG_SPEED := "ST00215_1_DB".RT01.JOG, VALUE_JOG_SPEED := "ST00215_1_DB".RT01_Speed.Jog, RAPID_STOP :=, RESET := #OPMODE.Reset, SPEED_DISPLAY_MODE := 2, MECHNICAL_FACTOR := 55.84, OPEN_BRAKE := "ST00215_1_DB".RT01.OPEN_BRAKE, VALUE_RAMP_UP := "RT_Standard_Ramp", VALUE_RAMP_DOWN := "RT_Standard_Ramp", IF_HMI := "GLOBAL_DRIVE_SEW_HMI_IF_DB".Drive[2], GENERAL_ALARM => "ST00215_1_DB".RT01_VFD01.GENERAL_ALARM, OUTPUT_STAGE_ENABLED => "ST00215_1_DB".RT01_VFD01.OUTPUT_STAGE_ENABLED, INVERTER_READY => "ST00215_1_DB".RT01_VFD01.INVERTER_READY, DRIVE_READY => "ST00215_1_DB".RT01_VFD01.DRIVE_READY, DRIVE_RUNNING => "ST00215_1_DB".RT01_VFD01.DRIVE_RUNNING, PARAMETER_2_SET =>)
   END_RUNG
   RUNG wire#powerrail
      Contact( "ST00215_1_DB".RT01.FORWARD )
      I_Contact( "ST00215_1_DB".RT01.REVERSE )
   END_RUNG wire#w1
   RUNG wire#powerrail
      I_Contact( "ST00215_1_DB".RT01.FORWARD )
      Contact( "ST00215_1_DB".RT01.REVERSE )
   END_RUNG wire#w2
   // the same network as SCL:
   "ST00215_RT01_VFD01_IDB"(PLANT_IDENTIFIER := WSTRING#'+ST00215.RT01-VFD01',   // "DRIVE_SEW_3PIO_PD_FB"
                           HARDWARE_OK := "OPMODE07_DB".HardwareOk.ST00215_RT01_VFD01,
                           SAFETY_OK := "IF_SAFE_TO_STND_DB".OPMode07.SafetyOK.ST00215_RT01,
                           HW_ID := "+ST00215_RT01-VFD01~FC_PD",
                           HEADUNIT_HW_ID := "+ST00215_RT01-VFD01~Movifit_Status",
                           SET_PARAMETER_2 := false,
                           CLOCKWISE_ROTATION := "ST00215_1_DB".RT01.FORWARD AND NOT "ST00215_1_DB".RT01.REVERSE,
                           COUNTERCLOCKWISE_ROTATION := NOT "ST00215_1_DB".RT01.FORWARD AND "ST00215_1_DB".RT01.REVERSE,
                           DIR_INDICATOR := 1,
                           FAST_SPEED := "ST00215_1_DB".RT01.FAST,
                           VALUE_FAST_SPEED := "ST00215_1_DB".RT01_Speed.Fast,
                           SLOW_SPEED := "ST00215_1_DB".RT01.SLOW,
                           VALUE_SLOW_SPEED := "ST00215_1_DB".RT01_Speed.Slow,
                           JOG_SPEED := "ST00215_1_DB".RT01.JOG,
                           VALUE_JOG_SPEED := "ST00215_1_DB".RT01_Speed.Jog,
                           RESET := #OPMODE.Reset,
                           SPEED_DISPLAY_MODE := 2,
                           MECHNICAL_FACTOR := 55.84,
                           OPEN_BRAKE := "ST00215_1_DB".RT01.OPEN_BRAKE,
                           VALUE_RAMP_UP := "RT_Standard_Ramp",
                           VALUE_RAMP_DOWN := "RT_Standard_Ramp",
                           IF_HMI := "GLOBAL_DRIVE_SEW_HMI_IF_DB".Drive[2],
                           GENERAL_ALARM => "ST00215_1_DB".RT01_VFD01.GENERAL_ALARM,
                           OUTPUT_STAGE_ENABLED => "ST00215_1_DB".RT01_VFD01.OUTPUT_STAGE_ENABLED,
                           INVERTER_READY => "ST00215_1_DB".RT01_VFD01.INVERTER_READY,
                           DRIVE_READY => "ST00215_1_DB".RT01_VFD01.DRIVE_READY,
                           DRIVE_RUNNING => "ST00215_1_DB".RT01_VFD01.DRIVE_RUNNING);
END_REGION
END_FUNCTION
